FUNCTION_BLOCK FB_Observable_BYTE EXTENDS FB_AbstractObservable
VAR
    _nVal:              BYTE;
    _nOldVal:           BYTE;
END_VAR

METHOD FB_init : BOOL
VAR_INPUT
    bInitRetains:       BOOL; // if TRUE, the retain variables are initialized (warm start / cold start)
    bInCopyCode:        BOOL;  // if TRUE, the instance afterwards gets moved into the copy code (online change)
    bAutoNotify:        BOOL;
END_VAR
THIS^._nTypeClass := __SYSTEM.TYPE_CLASS.TYPE_BYTE;
END_METHOD

PROPERTY nDataSize : UDINT
GET
nDataSize := SIZEOF(BYTE);
END_GET
END_PROPERTY

PROPERTY nValue8 : BYTE
GET
nValue8 := THIS^._nVal;
END_GET
SET
THIS^._nOldVal := THIS^._nVal;
THIS^._nVal := nValue8;

THIS^.NotifyWithConditions();
END_SET
END_PROPERTY

PROPERTY PROTECTED pData : POINTER TO BYTE
GET
pData := ADR(THIS^._nVal);
END_GET
END_PROPERTY

METHOD  ValueChanged : BOOL
VAR_INPUT
END_VAR
ValueChanged := THIS^._nOldVal <> THIS^._nVal;
END_METHOD

END_FUNCTION_BLOCK

(* stored: Version 1.1.0.1, ProductVersion 3.1.4024.12
   POU FB_Observable_BYTE: Id {b5a82f14-999a-0900-3426-ad6d97fd28ef}, SpecialFunc None
   Method FB_init: Id {ba6568d4-ed60-0181-3f0d-31118bec5235}
   Property nDataSize: Id {80114971-7e41-0759-3476-5e133361b4a9}
   Get Get: Id {9e1722d9-23fc-0a79-2350-6388f7356059}
   Property nValue8: Id {4328884a-5d6a-091b-24eb-52117cc5918f}
   Get Get: Id {311b7b1c-d65e-097b-1e50-15988af944da}
   Set Set: Id {7dc8ba13-55f6-0eb4-3f6c-f504a43d3da9}
   Property pData: Id {527767b2-d94a-0847-0124-7fa198f4aecf}
   Get Get: Id {e728a44a-8433-05a2-050e-09d05639d183}
   Method ValueChanged: Id {7ba15e8c-9027-0a10-3380-f3b900e45d25} *)
